// TIA Portal project "Proyecto3" (V14)

(* hardware
DEVICE "S71500/ET200MP station_1"  S7-1500 station
   slot 0: "Perfil soporte_0"  Rack  6ES7 590-1***0-0AA0
   slot 1: "PLC_1"  CPU 1511-1 PN  6ES7 511-1AK00-0AB0  V1.8
      slot 3: "Display de la CPU_1"  6ES7591-1AA00-0AA0
*)

// ===== PLC "PLC_1"  CPU 1511-1 PN =====

DATA_BLOCK "mis_datos"   // DB1
{ S7_Optimized_Access := 'TRUE' }
VERSION : 0.1
   VAR
      prueba : Bool;
      holaMundo : String := '¡Hell-o-Siemens!';
      contador : Int;
   END_VAR
BEGIN
END_DATA_BLOCK

DATA_BLOCK "OUTPUT"   // DB2
{ S7_Optimized_Access := 'FALSE' }
VERSION : 0.1
   VAR
      IN0 : Bool;   // *POSICIONAR POR TABLA
      IN1 : Bool;   // *POSICIONAR POR TABLA
      IN2 : Bool;   // *POSICIONAR POR TABLA
      IN3 : Bool;   // *POSICIONAR POR TABLA
      IN4 : Bool;   // *POSICIONAR POR TABLA
      IN5 : Bool;   // *POSICIONAR POR TABLA
      VACIO : Bool;
      VACIO_1 : Bool;
      HOLD : Bool;   // *PAUSAR
      SVON : Bool;   // *DAR PAR AL MOTOR
      DRIVE : Bool;   // *MUEVETE A POSICION POR TABLA (ON)
      RESET : Bool;   // *RESETEAR TABLA DE POSICION, INP, ALARMAS Y ORDENES
      SETUP : Bool;   // *VETE A ORIGEN
      "JOG-" : Bool;   // *MUEVETE A LA IZDA (DURANTE ON)
      "JOG+" : Bool;   // *MUEVETE A LA DRCHA (DURANTE ON)
      FLGTH : Bool;
      SPEED_RESTRICTION : Bool;
      MOVEMENT_MODE : Bool;
      SPEED : Bool;
      POSITION : Bool;   // *A ON ANTES DE "START_FLAG"
      ACCELERATION : Bool;
      DECELERATION : Bool;
      PUSHING_FORCE : Bool;
      TRIGGER_LV : Bool;
      PUSHING_SPEED : Bool;
      MOVING_FORCE : Bool;
      AREA_OUTPUT1 : Bool;
      AREA_OUTPUT2 : Bool;
      "TOLERANCE_RANGE_in position" : Bool;
      START_FLAG : Bool;   // *MUEVETE A POSICION POR MM (BIT 0 A ON)
      MOVEMENT_MODE_1 : Byte := 16#1;   // DEJAMOS EL BIT 0 A 1 PARA BALOR ABSOLUTO DE POSICION
      SPEED_byte : Int;
      POSITION_dword : DInt;   // *ESCRIBIR POSICIÓN POR MM
      ACCELERATION_word : Int;
      DECELERATION_word : Int;
      PUSHING_FORCE_word : Int;
      TRIGGER_LV_word : Int;
      PUSSING_SPEED_word : Int;
      MOVING_FORCE_word : Int;
      AREA1 : DInt;
      AREA2 : DInt;
      TOLERANCE_RANGE_dword : DInt;
      PILATZEN : Bool;
      PAKETATZEN : Bool;
      ETIKETATZEN : Bool;
      MENSAJE : Bool;
      CV_CONT1 : Int;
   END_VAR
BEGIN
END_DATA_BLOCK

DATA_BLOCK "MEMORIAS"   // DB3
{ S7_Optimized_Access := 'FALSE' }
VERSION : 0.1
   VAR
      INICIO_0 : Bool;
      INICIO_1 : Bool;
      INICIO_2 : Bool;
      INICIO_3 : Bool;
      INICIO_4 : Bool;
      INICIO_5 : Bool;
      INICIO_6 : Bool;
      M_EMERGENCIA : Bool;
      PROG_EMERGENCIA_0 : Bool;
      PROG_EMERGENCIA_1 : Bool;
      PROG_EMERGENCIA_2 : Bool;
      M_MANU_AUTO : Bool;
      M_C_UNICO : Bool;
      M_C_CONTINUO : Bool;
      M_REARME : Bool;
      M_PARO : Bool;
      M_POR_MM_0 : Bool;
      M_POR_MM_1 : Bool;
      M_POR_MM_2 : Bool;
      M_POR_MM_3 : Bool;
      FC_PILATU_0 : Bool;
      FC_PILATU_1 : Bool;
      FC_PILATU_2 : Bool;
      FC_PILATU_3 : Bool;
      PROGRAMA_0 : Bool;
      PROGRAMA_1 : Bool;
      PROGRAMA_2 : Bool;
      PROGRAMA_3 : Bool;
      PROGRAMA_4 : Bool;
      M_PAUSE : Bool;
      M_POSICION_PILATU : Byte;
      M_POSICION_ENPAKETATU : Byte;
      M_POSICION_ETIKETATU : Byte;
      FC_ENPAKETATU_0 : Bool;
      FC_ENPAKETATU_1 : Bool;
      FC_ENPAKETATU_2 : Bool;
      FC_ENPAKETATU_3 : Bool;
      FC_ETIKETATU_0 : Bool;
      FC_ETIKETATU_1 : Bool;
      FC_ETIKETATU_2 : Bool;
      FC_ETIKETATU_3 : Bool;
   END_VAR
BEGIN
END_DATA_BLOCK

DATA_BLOCK "INPUT"   // DB4
{ S7_Optimized_Access := 'FALSE' }
VERSION : 0.1
   VAR
      OUT0 : Bool;   // *POSICIÓN POR TABLA
      OUT1 : Bool;   // *POSICIÓN POR TABLA
      OUT2 : Bool;   // *POSICIÓN POR TABLA
      OUT3 : Bool;   // *POSICIÓN POR TABLA
      OUT4 : Bool;   // *POSICIÓN POR TABLA
      OUT5 : Bool;   // *POSICIÓN POR TABLA
      BUSY : Bool;   // *EN MOVIMIENTO
      SVRE : Bool;   // *MOTOR CON PAR
      SETON : Bool;   // *EN ORIGEN (ON)
      INP : Bool;   // *LLEGADA A POSICION (ON)
      AREA : Bool;
      WAREA : Bool;
      ESTOP : Bool;
      ALARM : Bool;   // *SI HAY ALARMA (ON)
      READY : Bool;   // *SIN ALARMA Y MOTOR CON PAR (ON)
      C_POSITION : DInt;   // *POSICION ACTUAL
      C_SPEED : Int;   // *VELOCIDAD ACTUAL
      C_PUSH_FORCE : Int;   // FUERZA ACTUAL
      TARGET_POSITION : DInt;
      ALARM1 : SInt;
      ALARM2 : SInt;
      ALARM3 : SInt;
      ALARM4 : SInt;
      MANU_AUTO : Bool;   // *PULSADORES WEB
      REARME : Bool;   // *PULSADORES WEB Y FISICO
      PARO : Bool;   // *PULSADORES WEB Y FISICO
      PAUSE : Bool;
      C_UNICO : Bool;   // *PULSADORES WEB
      C_CONTINUO : Bool;   // *PULSADORES WEB
      SETA : Bool;   // *PULSADORES WEB Y FISICO
      CONTINUAR : Bool;
      N_CICLOS : Int;   // *NUMEROS WEB
      POS_X_MM : DInt;   // *NUMEROS WEB
      POS_X_MM_ACEPTAR : Bool;   // *PULSADORES WEB
      WEB0 : Bool;   // *PULSADORES WEB
      WEB1 : Bool;   // *PULSADORES WEB
      WEB2 : Bool;   // *PULSADORES WEB
      WEB3 : Bool;   // *PULSADORES WEB
      WEB4 : Bool;   // *PULSADORES WEB
      WEB5 : Bool;   // *PULSADORES WEB
      WEB6 : Bool;   // *PULSADORES WEB
      WEB7 : Bool;   // *PULSADORES WEB
      WEB8 : Bool;   // *PULSADORES WEB
      WEB9 : Bool;   // *PULSADORES WEB
      WEB10 : Bool;   // *PULSADORES WEB
      "JOGWEB+" : Bool;
      "JOGWEB-" : Bool;
   END_VAR
BEGIN
END_DATA_BLOCK

ORGANIZATION_BLOCK "Main"   // OB1, LAD, ProgramCycle
TITLE = "Main Program Sweep (Cycle)"
{ S7_Optimized_Access := 'TRUE' }
VERSION : 0.1
   VAR_INPUT
      Initial_Call : Bool;   // Initial call of this OB
      Remanence : Bool;   // =True, if remanent data are available
   END_VAR
   VAR_TEMP
      Retorno : Int;
   END_VAR
BEGIN

REGION Network 1
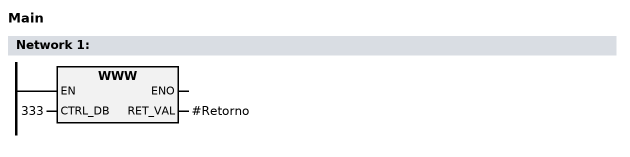
   #Retorno := WWW(CTRL_DB := 333);
END_REGION
END_ORGANIZATION_BLOCK